FUNCTION IrDistanceFromRaw : LREAL
VAR_INPUT
	rawValue : INT;
END_VAR
VAR
END_VAR

	IrDistanceFromRaw := 123.15 / EXPT( INT_TO_REAL(rawValue) * (10.0 / 32767.0), 1.119 );

END_FUNCTION

(* stored: Version 1.1.0.1, ProductVersion 3.1.4026.13
   POU IrDistanceFromRaw: Id {4b6affe3-0174-4995-bec2-7d9f1324cc0a}, SpecialFunc None *)
